PROGRAM MAIN
VAR
END_VAR

P_Dialog();

END_PROGRAM

(* stored: Version 1.1.0.1, ProductVersion 3.1.4022.16
   POU MAIN: Id {76b20082-c8a7-4433-ad64-571be51dcbfa}, SpecialFunc None *)
